TYPE ST_CalibrationStatus : STRUCT
    (* 已接受的标定请求编号。 *)
    nAcceptedRequestId : UDINT;
    (* 标定状态。 *)
    eState : E_CalibrationState;
    (* 标定是否完成。 *)
    bDone : BOOL;
    (* 标定是否发生错误。 *)
    bError : BOOL;
    (* 标定错误原因编号。 *)
    nErrorReason : UDINT;
    (* 生成的标定修订号。 *)
    nRevision : UDINT;
END_STRUCT
END_TYPE

(* stored: Version 1.1.0.1
   DUT ST_CalibrationStatus: Id {D3100000-0000-4000-8000-000000000029} *)
